PROGRAM P_DALI_Energy_Line2
VAR
	fbDALI_EnergyReporting: FB_DALI_EnergyReporting_Test;
	bReadEnergyData: BOOL;
	bCheckActiveEnergy	: BOOL;
END_VAR

VAR CONSTANT
	DALI_LINE_NUM: BYTE := 2;
END_VAR

fbDALI_EnergyReporting.ipDALICommunication := P_DALI_Background.arrfbKL6821Communication[DALI_LINE_NUM];

fbDALI_EnergyReporting(
	bExecute:= bReadEnergyData, 
	DALI_LINE_NUM:= DALI_LINE_NUM ,
	bCheckActiveEnergy := bCheckActiveEnergy,
	bBusy=> , 
	bActionBusy=> , 
	bErr=> , 
	nErrorId=> );

END_PROGRAM

(* stored: Version 1.1.0.1
   POU P_DALI_Energy_Line2: Id {93fae041-cb0d-4c1a-93c7-abaec0881fb9}, SpecialFunc None *)
